(* PLC project conveyor_management, Dassault Systèmes ControlBuild 2024x *)
(* stored: creationDateTime 2023-10-03T11:13:41-01:00 *)

FUNCTION_BLOCK bottling_line.conveyor_management
  VAR_INPUT
    productionRequest : BOOL := false;
  END_VAR
  VAR_INPUT
    pulseGenerator : BOOL := false;
    bottleFilled : BOOL := false;
    bottlePresent : BOOL := false;
  END_VAR
  VAR_OUTPUT
    load : BOOL := false;
    evacuate : BOOL := false;
    convoy : BOOL := false;
  END_VAR
  VAR_OUTPUT
    valve5 : BOOL := false;
  END_VAR
  VAR
    encoder : INT := 0;
  END_VAR
  VAR CONSTANT
    value : INT := 10;
    increment : INT := 1;
  END_VAR

INITIAL_STEP 10:
  10_INLINE1(N);
  COMPUTE_FUNCTION_BLOCKS(S);
END_STEP
ACTION 10_INLINE1:
  encoder := 0;
END_ACTION
TRANSITION FROM 10 TO 11
  := productionRequest AND bottlePresent;
END_TRANSITION
TRANSITION FROM 10 TO 12
  := productionRequest AND NOT bottlePresent;
END_TRANSITION
STEP 11:
  11_INLINE2(N);
END_STEP
ACTION 11_INLINE2:
  valve5;
END_ACTION
TRANSITION FROM 11 TO 12
  := bottleFilled;
END_TRANSITION
STEP 12:
  12_INLINE3(N);
END_STEP
ACTION 12_INLINE3:
  load := TRUE;
  evacuate := TRUE;
END_ACTION
TRANSITION FROM 12 TO 13
  := T/X12/2 s;
END_TRANSITION
STEP 13:
  13_INLINE4(N);
END_STEP
ACTION 13_INLINE4:
  load := FALSE;
  evacuate := FALSE;
END_ACTION
TRANSITION FROM 13 TO 14
  := T/X13/2 s;
END_TRANSITION
STEP 14:
  14_INLINE5(N);
END_STEP
ACTION 14_INLINE5:
  convoy;
  IF RE pulseGenerator  THEN encoder := encoder + increment;
  END_IF;
END_ACTION
TRANSITION FROM 14 TO 10
  := (encoder >= value);
END_TRANSITION
ACTION COMPUTE_FUNCTION_BLOCKS:  (* blocks drawn on the SFC sheet *)
  G1:
END_ACTION
END_FUNCTION_BLOCK
